% RSLogix 500 project I2P JOB 8 Brandon F.RSS, saved by version 10.00.00.00 %
PROJECT "ML05B"    % processor: Bul.1763 MicroLogix 1100 Series B %

PROGRAM FILES
  LAD 2   5 rungs

DATA FILES
  O0 OUTPUT  4 elements
  I1 INPUT  6 elements
  S2 STATUS  66 elements
  B3 BINARY  1 elements
  T4 TIMER  1 elements
  C5 COUNTER  1 elements
  R6 CONTROL  1 elements
  N7 INTEGER  1 elements
  F8 FLOAT  1 elements

LADDER 2
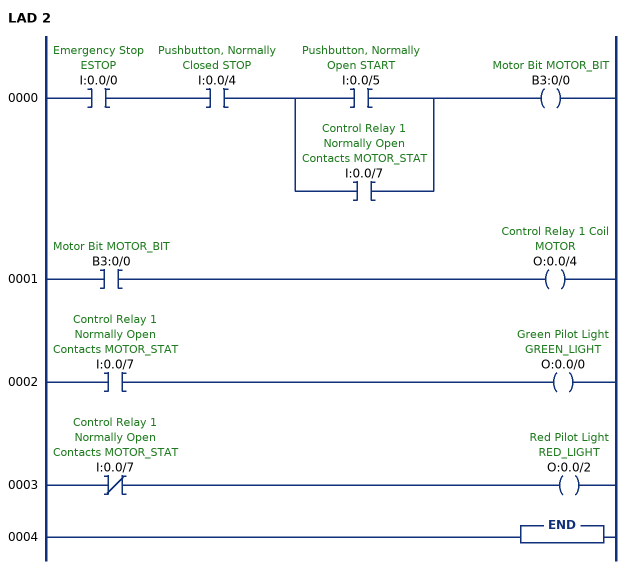
% Rung: 0 %
SOR XIC I:0.0/0 XIC I:0.0/4 BST XIC I:0.0/5 NXB XIC I:0.0/7 BND OTE B3:0/0 EOR
%   I:0.0/0  ESTOP  "Emergency Stop" %
%   I:0.0/4  STOP  "Pushbutton, Normally Closed" %
%   I:0.0/5  START  "Pushbutton, Normally Open" %
%   I:0.0/7  MOTOR_STAT  "Control Relay 1 Normally Open Contacts" %
%   B3:0/0  MOTOR_BIT  "Motor Bit" %
% Rung: 1 %  % edit flag set %
SOR XIC B3:0/0 OTE O:0.0/4 EOR
%   B3:0/0  MOTOR_BIT  "Motor Bit" %
%   O:0.0/4  MOTOR  "Control Relay 1 Coil" %
% Rung: 2 %
SOR XIC I:0.0/7 OTE O:0.0/0 EOR
%   I:0.0/7  MOTOR_STAT  "Control Relay 1 Normally Open Contacts" %
%   O:0.0/0  GREEN_LIGHT  "Green Pilot Light" %
% Rung: 3 %
SOR XIO I:0.0/7 OTE O:0.0/2 EOR
%   I:0.0/7  MOTOR_STAT  "Control Relay 1 Normally Open Contacts" %
%   O:0.0/2  RED_LIGHT  "Red Pilot Light" %
% Rung: 4 %
SOR END EOR
